{attribute 'qualified_only'}
VAR_GLOBAL
	stBoxParam : ST_BoxParam;
END_VAR

(* stored: Version 1.1.0.1, ProductVersion 3.1.4024.12
   GVL Parameters: Id {fa2216f4-7237-4717-a395-6c1475299f72} *)
